// TIA Portal V20 export
TYPE "HMI_TimeSwitch"
   STRUCT
      DwCurr { ExternalWritable := 'False'} : Int;   // Currently used day of the week
      TdCurr { ExternalWritable := 'False'} : DInt;   // Currently used time of the day
      StCurr { ExternalWritable := 'False'} : Bool;   // Current daylight saving time
      DwAs { ExternalWritable := 'False'} : Int;   // AS day of the week
      TdAs { ExternalWritable := 'False'} : DInt;   // AS time of the day
      DwLoc { ExternalWritable := 'False'} : Int;   // Local day of the week
      TdLoc { ExternalWritable := 'False'} : DInt;   // Local time of the day
      StLoc { ExternalWritable := 'False'} : Bool;   // Local daylight saving time active
      DwExt { ExternalWritable := 'False'} : Int;   // External day of the week
      TdExt { ExternalWritable := 'False'} : DInt;   // External time of the day
      StExt { ExternalWritable := 'False'} : Bool;   // External daylight saving time active / Local daylight saving time active
      TiExtQc { ExternalWritable := 'False'} : Byte := BYTE#16#80;   // Quality of external time signal
      P_Time : Real := 2.0;   // Time for on/off pulse
      OnOp : Bool;   // 1=On Mode: On Mode by Operator
      OosOP : Bool;   // 1=Oos Mode: Oos Mode by Operator
      On { ExternalWritable := 'False'} : Bool;   // Output switch point general
      P_On { ExternalWritable := 'False'} : Bool;   // On pulse output switch point general
      P_Off { ExternalWritable := 'False'} : Bool;   // Off pulse output sitch point general
      NxTiOn { ExternalWritable := 'False'} : Real;   // Next on switch point
      NxTiOff { ExternalWritable := 'False'} : Real;   // Next off switch point
      On1 { ExternalWritable := 'False'} : Bool;   // Output switch point 1
      P_On1 { ExternalWritable := 'False'} : Bool;   // On pulse output switch point 1
      P_Off1 { ExternalWritable := 'False'} : Bool;   // Off pulse output sitch point 1
      NxTiOn1 { ExternalWritable := 'False'} : Real;   // Next on switch point
      NxTiOff1 { ExternalWritable := 'False'} : Real;   // Next off switch point
      SwTiOn1 : DInt;   // time switching point 1 on
      SwTiOff1 : DInt := DINT#86399;   // time switching point 1 off
      SwAct1 : Byte;   // active days switching point 1
      On2 { ExternalWritable := 'False'} : Bool;   // Output switch point 2
      P_On2 { ExternalWritable := 'False'} : Bool;   // On pulse output switch point 2
      P_Off2 { ExternalWritable := 'False'} : Bool;   // Off pulse output sitch point 2
      NxTiOn2 { ExternalWritable := 'False'} : Real;   // Next on switch point
      NxTiOff2 { ExternalWritable := 'False'} : Real;   // Next off switch point
      SwTiOn2 : DInt;   // time switching point 2 on
      SwTiOff2 : DInt := DINT#86399;   // time switching point 2 off
      SwAct2 : Byte;   // active days switching point 2
      On3 { ExternalWritable := 'False'} : Bool;   // Output switch point 3
      P_On3 { ExternalWritable := 'False'} : Bool;   // On pulse output switch point 3
      P_Off3 { ExternalWritable := 'False'} : Bool;   // Off pulse output sitch point 3
      NxTiOn3 { ExternalWritable := 'False'} : Real;   // Next on switch point
      NxTiOff3 { ExternalWritable := 'False'} : Real;   // Next off switch point
      SwTiOn3 : DInt;   // time switching point 3 on
      SwTiOff3 : DInt := DINT#86399;   // time switching point 3 off
      SwAct3 : Byte;   // active days switching point 3
      On4 { ExternalWritable := 'False'} : Bool;   // Output switch point 4
      P_On4 { ExternalWritable := 'False'} : Bool;   // On pulse output switch point 4
      P_Off4 { ExternalWritable := 'False'} : Bool;   // Off pulse output sitch point 4
      NxTiOn4 { ExternalWritable := 'False'} : Real;   // Next on switch point
      NxTiOff4 { ExternalWritable := 'False'} : Real;   // Next off switch point
      SwTiOn4 : DInt;   // time switching point 4 on
      SwTiOff4 : DInt := DINT#86399;   // time switching point 4 off
      SwAct4 : Byte;   // active days switching point 4
      On5 { ExternalWritable := 'False'} : Bool;   // Output switch point 5
      P_On5 { ExternalWritable := 'False'} : Bool;   // On pulse output switch point 5
      P_Off5 { ExternalWritable := 'False'} : Bool;   // Off pulse output sitch point 5
      NxTiOn5 { ExternalWritable := 'False'} : Real;   // Next on switch point
      NxTiOff5 { ExternalWritable := 'False'} : Real;   // Next off switch point
      SwTiOn5 : DInt;   // time switching point 5 on
      SwTiOff5 : DInt := DINT#86399;   // time switching point 5 off
      SwAct5 : Byte;   // active days switching point 5
      On6 { ExternalWritable := 'False'} : Bool;   // Output switch point 6
      P_On6 { ExternalWritable := 'False'} : Bool;   // On pulse output switch point 6
      P_Off6 { ExternalWritable := 'False'} : Bool;   // Off pulse output sitch point 6
      NxTiOn6 { ExternalWritable := 'False'} : Real;   // Next on switch point
      NxTiOff6 { ExternalWritable := 'False'} : Real;   // Next off switch point
      SwTiOn6 : DInt;   // time switching point 6 on
      SwTiOff6 : DInt := DINT#86399;   // time switching point 6 off
      SwAct6 : Byte;   // active days switching point 6
      On7 { ExternalWritable := 'False'} : Bool;   // Output switch point 7
      P_On7 { ExternalWritable := 'False'} : Bool;   // On pulse output switch point 7
      P_Off7 { ExternalWritable := 'False'} : Bool;   // Off pulse output sitch point 7
      NxTiOn7 { ExternalWritable := 'False'} : Real;   // Next on switch point
      NxTiOff7 { ExternalWritable := 'False'} : Real;   // Next off switch point
      SwTiOn7 : DInt;   // time switching point 7 on
      SwTiOff7 : DInt := DINT#86399;   // time switching point 7 off
      SwAct7 : Byte;   // active days switching point 7
      On8 { ExternalWritable := 'False'} : Bool;   // Output switch point 8
      P_On8 { ExternalWritable := 'False'} : Bool;   // On pulse output switch point 8
      P_Off8 { ExternalWritable := 'False'} : Bool;   // Off pulse output sitch point 8
      NxTiOn8 { ExternalWritable := 'False'} : Real;   // Next on switch point
      NxTiOff8 { ExternalWritable := 'False'} : Real;   // Next off switch point
      SwTiOn8 : DInt;   // time switching point 8 on
      SwTiOff8 : DInt := DINT#86399;   // time switching point 8 off
      SwAct8 : Byte;   // active days switching point 8
      Status1 { ExternalWritable := 'False'} : DWord;   // Status word 1, defined in the online help
      Status2 { ExternalWritable := 'False'} : DWord;   // Status word 2, defined in the online help
      Status3 { ExternalWritable := 'False'} : DWord;   // Status word 3, defined in the online help
      Status4 { ExternalWritable := 'False'} : DWord;   // Status word 4, defined in the online help
      OS_PermOut { ExternalWritable := 'False'} : DWord := DWORD#16#FFFF_FFFF;   // Display of operator permissions OS_Perm
      OS_PermLog { ExternalWritable := 'False'} : DWord := DWORD#16#FFFF_FFFF;   // Operator permissions with settings changed by the block algorithm
      ST_Worst { ExternalWritable := 'False'} : Byte := BYTE#16#80;   // Worst signal status
      AlarmState { ExternalWritable := 'False'} : Word;   // Alarm Status for group display
   END_STRUCT;
END_TYPE
